(* Logix 5000 project; controller OT8 vendor 1 type 14 code 149 rev 32.11; software revision 32.04 *)

TASK MainTask (continuous, watchdog 500 ms) : MainProgram

MODULES
   Local : vendor 1 type 14 code 149 (Compact 0, rev 32.11)
      Discrete_IO : Embedded (Compact 1, rev 3.1, Output RPI 20 ms)
      VFD0602 : PowerFlex 525-EENET (Ethernet 100.100.100.11, rev 7.1, Output RPI 20 ms)
      VFD0543 : PowerFlex 525-EENET (Ethernet 100.100.100.10, rev 7.1, Output RPI 20 ms)
      VFD0643 : PowerFlex 525-EENET (Ethernet 100.100.100.12, rev 7.1, Output RPI 20 ms)
END_MODULES

TYPE VFD_CONTROL :
STRUCT
   START_CONDITION : BOOL;   // START CONDITIONS TRUE
   AUTO_RUN_VFD : BOOL;   // RUN VFD IN AUTO MODE
   VFD_RUNNING : BOOL;
   ALARM : BOOL;   // VFD ALARM WENT ACTIVE
   VFD_RUN_REFERENCE : REAL;   // VFD SPEED REFERENCE TO RUN
   SELECTION_SPEEDS_STORAGE : REAL[17];   // VFD STORED SPEED
   START_TIMER : TIMER;   // VFD START DELAY TIMER READY TO START
   VFD_FP : VFD_FACEPLATE_DATA;
   ALARM_LATCH : BOOL;   // LOCAL ROUTINE ALARM LATCH
END_STRUCT
END_TYPE

TYPE VFD_FACEPLATE_DATA :
STRUCT
   _0 : BOOL;   // HMI FACEPLATE SPEED CHANGE
   _1 : BOOL;   // HMI FACEPLATE DISCONNECT ON
   _2 : BOOL;   // HMI FACEPLATE DISCONNECT FAULTED
   _3 : BOOL;   // HMI FACEPLATE MCP FAULTED
   _4 : BOOL;   // HMI FACEPLATE VFD READY
   _5 : BOOL;   // HMI FACEPLATE VFD FAULTED
   _6 : BOOL;   // HMI FACEPLATE ACTIVE
   _7 : BOOL;   // HMI FACEPLATE VFD COMMS OK
   _8 : BOOL;   // HMI FACEPLATE JOG PB
   _9 : BOOL;   // HMI FACEPLATE JOGGING INDICATOR
   _10 : BOOL;   // HMI FACEPLATE SPARE At Reference Reached (latching)
   _11 : BOOL;   // HMI FACEPLATE AUTO ACTIVE
   _12 : BOOL;   // HMI FACEPLATE MANUAL RUN MODE ACTIVE
   SPARE1 : BOOL;
   SPARE2 : BOOL;
   SPARE3 : BOOL;
   HMI_SPEED_REF : REAL;   // VFD SPEED REFERENCE FROM HMI
   HMI_OUT_FREQ : REAL;   // VFD OUTPUT FREQUENCY TO HMI
   HMI_OUT_CUR : REAL;   // VFD OUTPUT CURRENT TO HMI
   SPEED_REF : REAL;   // VFD SELECTED SPEED REFERENCE
   COMMS_FAULT_CODE : DINT;   // .2 AND .9 HIGH = COMMS GOOD
END_STRUCT
END_TYPE

VAR_GLOBAL   (* controller tags *)
   ALARM_ACTIVE : BOOL;   // LINE 41 PLC ALARM BIT IS SET
   ALARMS : DINT[3];
        [0]   // VFD ALARMS
        [0].0   // VFD0543 NOT READY ALARM
        [0].1   // VFD0602 NOT READY ALARM
        [0].10   // VFD1043 NOT READY ALARM
        [0].11   // VFD1102 NOT READY ALARM
        [0].12   // VFD1143 NOT READY ALARM
        [0].13   // VFD1202 NOT READY ALARM
        [0].14   // VFD1243 NOT READY ALARM
        [0].2   // VFD0643 NOT READY ALARM
        [0].3   // VFD0702 NOT READY ALARM
        [0].4   // VFD0743 NOT READY ALARM
        [0].5   // VFD0802 NOT READY ALARM
        [0].6   // VFD0843 NOT READY ALARM
        [0].7   // VFD0902 NOT READY ALARM
        [0].8   // VFD0943 NOT READY ALARM
        [0].9   // VFD1002 NOT READY ALARM
        [1]   // DISC ALARMS
        [1].0   // DS0543 AUX CONTACT ALARM
        [1].1   // DS0602 AUX CONTACT ALARM
        [1].10   // DS1043 AUX CONTACT ALARM
        [1].11   // DS1102 AUX CONTACT ALARM
        [1].12   // DS1143 AUX CONTACT ALARM
        [1].13   // DS1202 AUX CONTACT ALARM
        [1].14   // DS1243 AUX CONTACT ALARM
        [1].2   // DS0643 AUX CONTACT ALARM
        [1].3   // DS0702 AUX CONTACT ALARM
        [1].4   // DS0743 AUX CONTACT ALARM
        [1].5   // DS0802 AUX CONTACT ALARM
        [1].6   // DS0808 AUX CONTACT ALARM
        [1].7   // DS0814 AUX CONTACT ALARM
        [1].8   // DS0943 AUX CONTACT ALARM
        [1].9   // DS1002 AUX CONTACT ALARM
        [2]   // E-STOP ALARMS
        [2].0   // E-STOP MAIN ENCLOSURE PBLT1402 ALARM
        [2].1   // E-STOP REMOTE #1 PBLT1404 ALARM
        [2].2   // E-STOP REMOTE #2 PBLT1406 ALARM
        [2].3   // E-STOP REMOTE #3 PBLT1408 ALARM
        [2].4   // E-STOP REMOTE #4 PBLT1410 ALARM
        [2].5   // E-STOP REMOTE #5PBLT1412 ALARM
        [2].6   // E-STOP REMOTE #6 PBLT1414 ALARM
   DS0543 : ALIAS FOR Local:1:I.Data.8;   // DS0543 AUX CONTACT
   DS0602 : ALIAS FOR Local:1:I.Data.9;   // DS0602 AUX CONTACT
   DS0643 : ALIAS FOR Local:1:I.Data.10;   // DS0643 AUX CONTACT
   LINE_100_RESET : ALIAS FOR Local:1:I.Data.6;   // LINE 100 RESET ALARMS
   LINE_100_RUN_MODE_ACTIVE : BOOL := 1;   // LINE 100 RUN MODE ACTIVE
   LINE_100_RUN_MODE_READY : BOOL := 1;   // LINE 100 IS READY TO START
   LINE_100_STARTUP_ANNUNCIATION_DELAY : TIMER := (PRE := 3000);   // LINE 100 STARTUP DELAY
   LINE_100_VFD_READY : BOOL := 1;   // LINE 100 VFDS READY
   LINE_200_RUN_MODE_ACTIVE : BOOL := 1;   // LINE 200 RUN MODE ACTIVE
   LINE_200_RUN_MODE_READY : BOOL := 1;   // LINE 200 IS READY TO START
   LINE_200_START_FLASH_BIT : BOOL;   // BIT TO FLASH LINE 200 START PB PILOT LIGHT DURING STARTUP
   LINE_200_STARTUP_ANNUNCIATION_DELAY : TIMER := (PRE := 3000);   // LINE 200 STARTUP DELAY
   LINE_200_VFD_READY : BOOL := 1;   // LINE 200 VFD READY
   LINE_200_VFDS_READY : BOOL;   // LINE 200 VFDS READY
   PB1831 : ALIAS FOR Local:1:I.Data.2;   // LINE 100 STOP PB
   PB1832 : ALIAS FOR Local:1:I.Data.3;   // LINE 100 START PB
   PB1833 : ALIAS FOR Local:1:I.Data.4;   // LINE 200 STOP PB
   PB1834 : ALIAS FOR Local:1:I.Data.5;   // LINE 200 START PB
   PBLT1832 : ALIAS FOR Local:1:O.Data.0;   // LINE 100 START PB PILOT LIGHT
   PBLT1834 : ALIAS FOR Local:1:O.Data.1;   // LINE 200 START PB PILOT LIGHT
   SAFETY_RELAY_RESET_ONS : BOOL;
   SR1426 : ALIAS FOR Local:1:I.Data.0;   // LINE 200 SAFETY RELAY
   SR1526 : ALIAS FOR Local:1:I.Data.1;   // LINE 100 SAFETY RELAY
   STARTUP_ANNUNCIATION_DELAY : TIMER;   // STARTUP ANNUCIATION TIMER
   SYSTEM_AUTO_RUN_MODE_ACTIVE : BOOL;   // RUN MODE ACTIVE
   SYSTEM_AUTO_RUN_MODE_READY : BOOL;   // SYSTEM READY TO ENTER AUTO RUN MODE
   SYSTEM_FLASH_BIT : BOOL := 1;   // FLASH BIT
   SYSTEM_FLASHER_OFF_TIME : TIMER := (PRE := 500, ACC := 500);   // SYSTEM FLASHER OFF TIME
   SYSTEM_FLASHER_ON_TIME : TIMER := (PRE := 500, ACC := 19, EN := 1, TT := 1);   // SYSTEM FLASHER ON TIME
   VFD0543 : VFD_CONTROL := (START_CONDITION := 1, START_TIMER.PRE := 500, START_TIMER.ACC := 500, START_TIMER.EN := 1, START_TIMER.DN := 1);
   VFD0602 : VFD_CONTROL := (START_CONDITION := 1, START_TIMER.PRE := 500, START_TIMER.ACC := 500, START_TIMER.EN := 1, START_TIMER.DN := 1);
   VFD0643 : VFD_CONTROL := (START_CONDITION := 1, START_TIMER.EN := 1, START_TIMER.DN := 1);
END_VAR

PROGRAM MainProgram   (* main routine MainRoutine *)
VAR
   AFI : DINT;
   PBLT1437 : ALIAS FOR Local:1:I.Data.6;   // RESET PUSHBUTTON LINE 200
   PBLT1537 : ALIAS FOR Local:1:I.Data.7;   // RESET PUSHBUTTON LINE 100
END_VAR

ROUTINE ALARMS   (* ladder *)
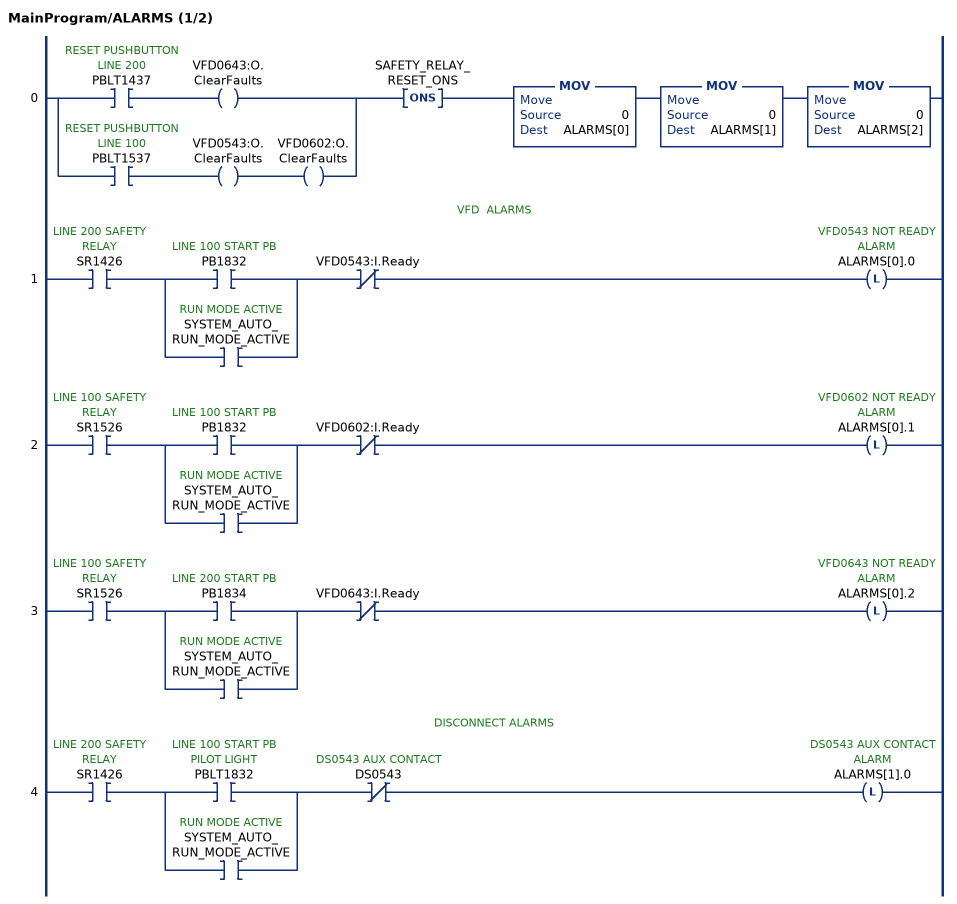
   0: [XIC(PBLT1437) OTE(VFD0643:O.ClearFaults) ,XIC(PBLT1537) OTE(VFD0543:O.ClearFaults) OTE(VFD0602:O.ClearFaults) ]ONS(SAFETY_RELAY_RESET_ONS)MOV(0,ALARMS[0])MOV(0,ALARMS[1])MOV(0,ALARMS[2]);
   // VFD  ALARMS
   1: XIC(SR1426)[XIC(PB1832) ,XIC(SYSTEM_AUTO_RUN_MODE_ACTIVE) ]XIO(VFD0543:I.Ready)OTL(ALARMS[0].0);
   2: XIC(SR1526)[XIC(PB1832) ,XIC(SYSTEM_AUTO_RUN_MODE_ACTIVE) ]XIO(VFD0602:I.Ready)OTL(ALARMS[0].1);
   3: XIC(SR1526)[XIC(PB1834) ,XIC(SYSTEM_AUTO_RUN_MODE_ACTIVE) ]XIO(VFD0643:I.Ready)OTL(ALARMS[0].2);
   // DISCONNECT ALARMS
   4: XIC(SR1426)[XIC(PBLT1832) ,XIC(SYSTEM_AUTO_RUN_MODE_ACTIVE) ]XIO(DS0543)OTL(ALARMS[1].0);
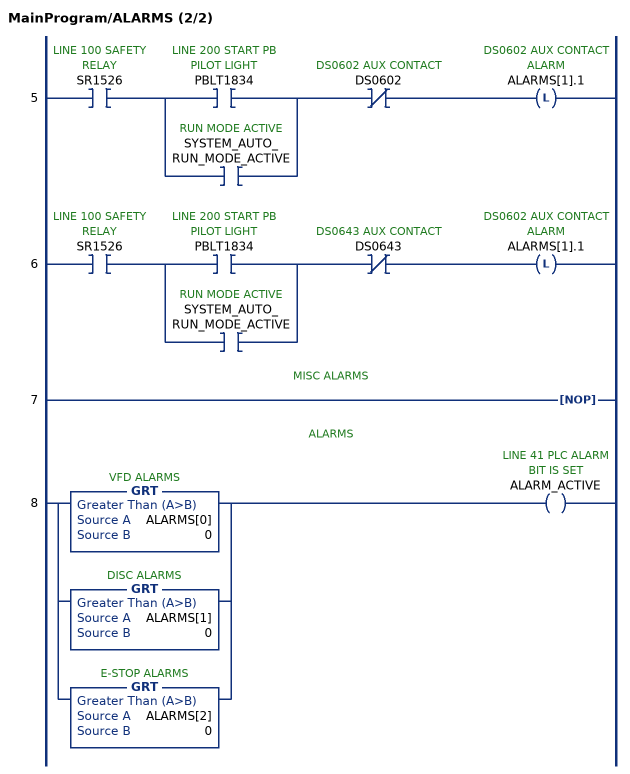
   5: XIC(SR1526)[XIC(PBLT1834) ,XIC(SYSTEM_AUTO_RUN_MODE_ACTIVE) ]XIO(DS0602)OTL(ALARMS[1].1);
   6: XIC(SR1526)[XIC(PBLT1834) ,XIC(SYSTEM_AUTO_RUN_MODE_ACTIVE) ]XIO(DS0643)OTL(ALARMS[1].1);
   // MISC ALARMS
   7: NOP();
   // ALARMS
   8: [GRT(ALARMS[0],0) ,GRT(ALARMS[1],0) ,GRT(ALARMS[2],0) ]OTE(ALARM_ACTIVE);
END_ROUTINE

ROUTINE MainRoutine   (* ladder *)
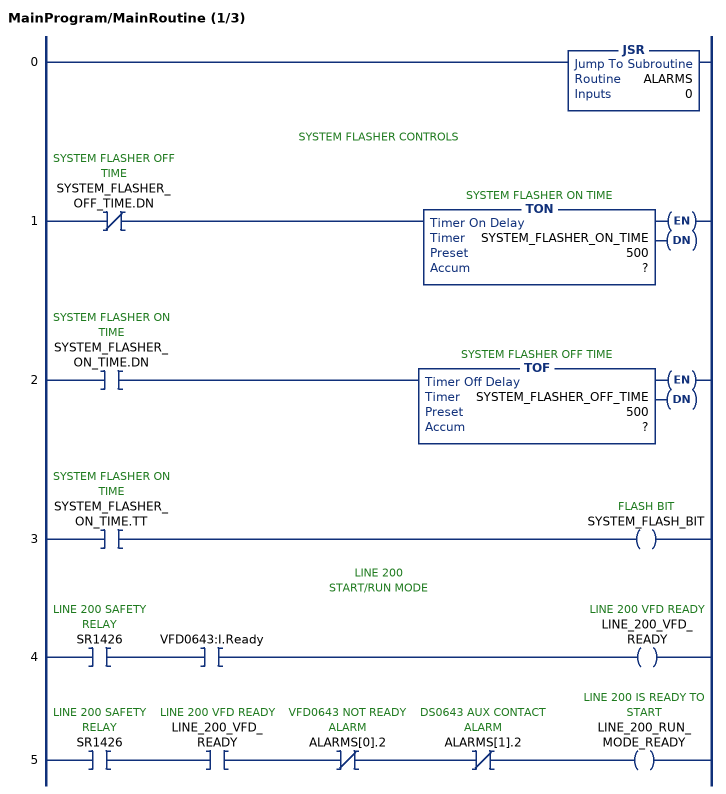
   0: JSR(ALARMS,0);
   // SYSTEM FLASHER CONTROLS
   1: XIO(SYSTEM_FLASHER_OFF_TIME.DN)TON(SYSTEM_FLASHER_ON_TIME,?,?);
   2: XIC(SYSTEM_FLASHER_ON_TIME.DN)TOF(SYSTEM_FLASHER_OFF_TIME,?,?);
   3: XIC(SYSTEM_FLASHER_ON_TIME.TT)OTE(SYSTEM_FLASH_BIT);
   // LINE 200
   // START/RUN MODE
   4: XIC(SR1426)XIC(VFD0643:I.Ready)OTE(LINE_200_VFD_READY);
   5: XIC(SR1426)XIC(LINE_200_VFD_READY)XIO(ALARMS[0].2)XIO(ALARMS[1].2)OTE(LINE_200_RUN_MODE_READY);
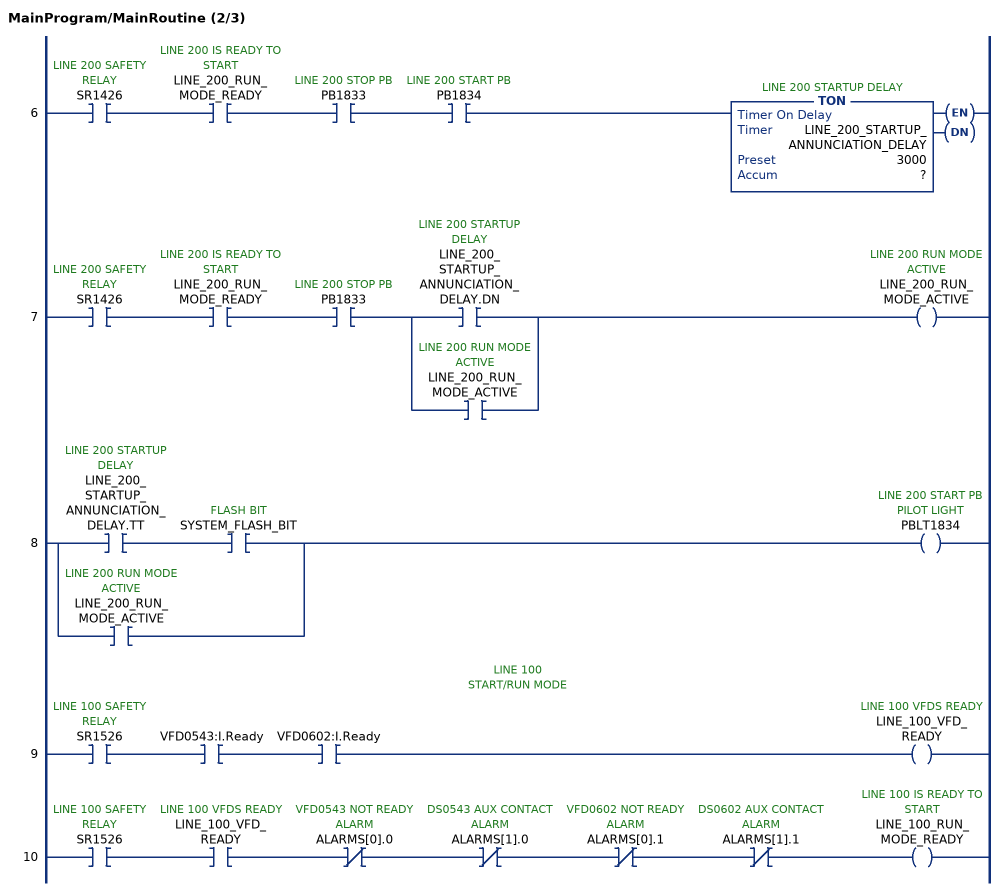
   6: XIC(SR1426)XIC(LINE_200_RUN_MODE_READY)XIC(PB1833)XIC(PB1834)TON(LINE_200_STARTUP_ANNUNCIATION_DELAY,?,?);
   7: XIC(SR1426)XIC(LINE_200_RUN_MODE_READY)XIC(PB1833)[XIC(LINE_200_STARTUP_ANNUNCIATION_DELAY.DN) ,XIC(LINE_200_RUN_MODE_ACTIVE) ]OTE(LINE_200_RUN_MODE_ACTIVE);
   8: [XIC(LINE_200_STARTUP_ANNUNCIATION_DELAY.TT) XIC(SYSTEM_FLASH_BIT) ,XIC(LINE_200_RUN_MODE_ACTIVE) ]OTE(PBLT1834);
   // LINE 100
   // START/RUN MODE
   9: XIC(SR1526)XIC(VFD0543:I.Ready)XIC(VFD0602:I.Ready)OTE(LINE_100_VFD_READY);
   10: XIC(SR1526)XIC(LINE_100_VFD_READY)XIO(ALARMS[0].0)XIO(ALARMS[1].0)XIO(ALARMS[0].1)XIO(ALARMS[1].1)OTE(LINE_100_RUN_MODE_READY);
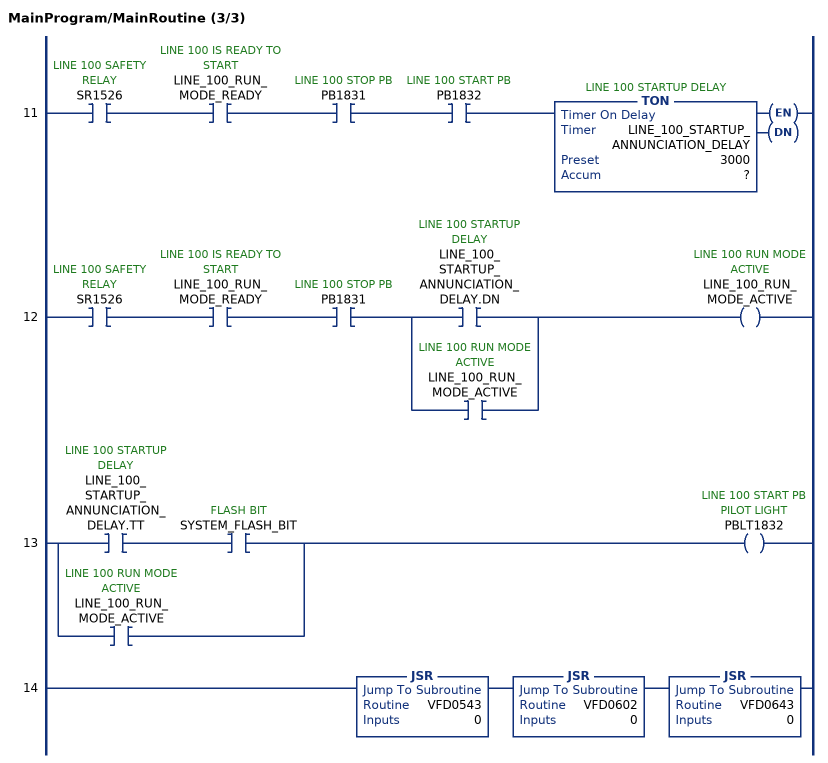
   11: XIC(SR1526)XIC(LINE_100_RUN_MODE_READY)XIC(PB1831)XIC(PB1832)TON(LINE_100_STARTUP_ANNUNCIATION_DELAY,?,?);
   12: XIC(SR1526)XIC(LINE_100_RUN_MODE_READY)XIC(PB1831)[XIC(LINE_100_STARTUP_ANNUNCIATION_DELAY.DN) ,XIC(LINE_100_RUN_MODE_ACTIVE) ]OTE(LINE_100_RUN_MODE_ACTIVE);
   13: [XIC(LINE_100_STARTUP_ANNUNCIATION_DELAY.TT) XIC(SYSTEM_FLASH_BIT) ,XIC(LINE_100_RUN_MODE_ACTIVE) ]OTE(PBLT1832);
   14: JSR(VFD0543,0)JSR(VFD0602,0)JSR(VFD0643,0);
END_ROUTINE

ROUTINE VFD0543   (* ladder *)
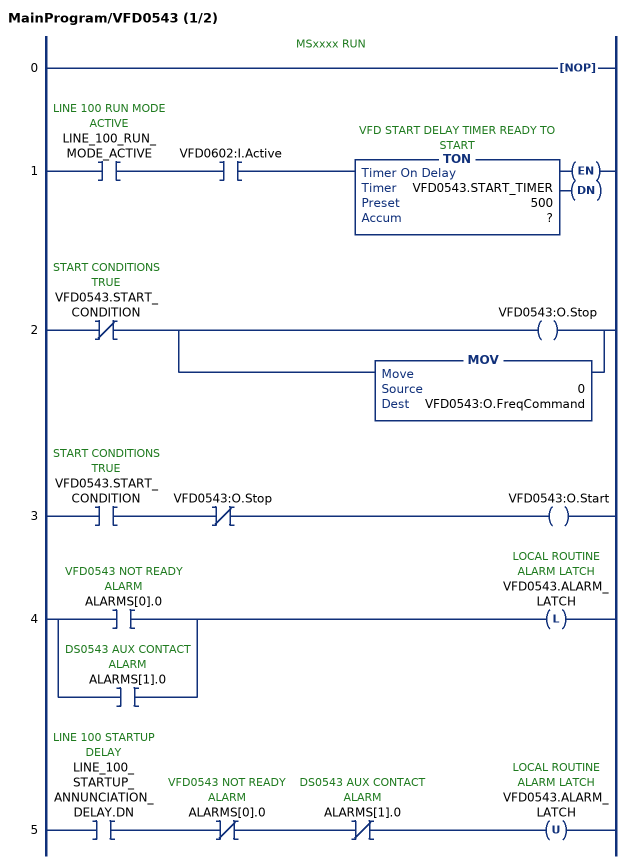
   // MSxxxx RUN
   0: NOP();
   1: XIC(LINE_100_RUN_MODE_ACTIVE)XIC(VFD0602:I.Active)TON(VFD0543.START_TIMER,?,?);
   2: XIO(VFD0543.START_CONDITION)[OTE(VFD0543:O.Stop) ,MOV(0,VFD0543:O.FreqCommand) ];
   3: XIC(VFD0543.START_CONDITION)XIO(VFD0543:O.Stop)OTE(VFD0543:O.Start);
   4: [XIC(ALARMS[0].0) ,XIC(ALARMS[1].0) ]OTL(VFD0543.ALARM_LATCH);
   5: XIC(LINE_100_STARTUP_ANNUNCIATION_DELAY.DN)XIO(ALARMS[0].0)XIO(ALARMS[1].0)OTU(VFD0543.ALARM_LATCH);
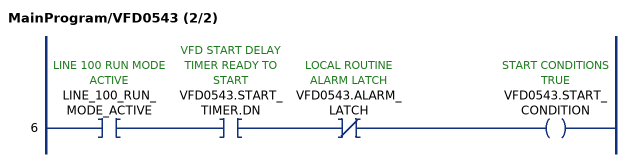
   6: XIC(LINE_100_RUN_MODE_ACTIVE)XIC(VFD0543.START_TIMER.DN)XIO(VFD0543.ALARM_LATCH)OTE(VFD0543.START_CONDITION);
END_ROUTINE

ROUTINE VFD0602   (* ladder *)
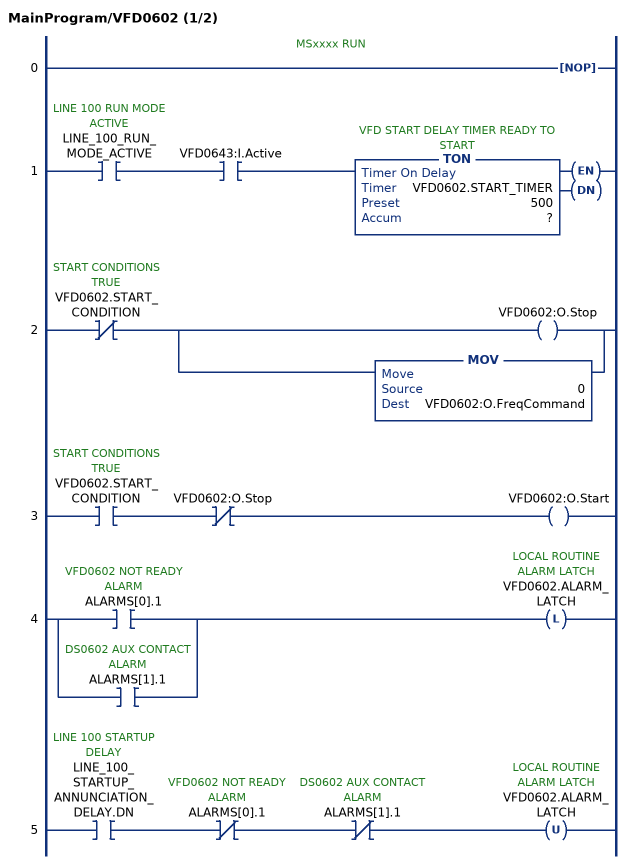
   // MSxxxx RUN
   0: NOP();
   1: XIC(LINE_100_RUN_MODE_ACTIVE)XIC(VFD0643:I.Active)TON(VFD0602.START_TIMER,?,?);
   2: XIO(VFD0602.START_CONDITION)[OTE(VFD0602:O.Stop) ,MOV(0,VFD0602:O.FreqCommand) ];
   3: XIC(VFD0602.START_CONDITION)XIO(VFD0602:O.Stop)OTE(VFD0602:O.Start);
   4: [XIC(ALARMS[0].1) ,XIC(ALARMS[1].1) ]OTL(VFD0602.ALARM_LATCH);
   5: XIC(LINE_100_STARTUP_ANNUNCIATION_DELAY.DN)XIO(ALARMS[0].1)XIO(ALARMS[1].1)OTU(VFD0602.ALARM_LATCH);
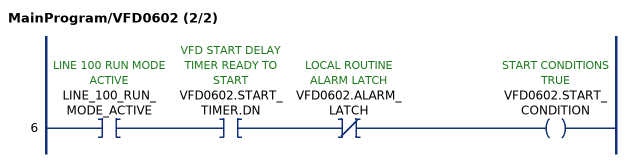
   6: XIC(LINE_100_RUN_MODE_ACTIVE)XIC(VFD0602.START_TIMER.DN)XIO(VFD0602.ALARM_LATCH)OTE(VFD0602.START_CONDITION);
END_ROUTINE

ROUTINE VFD0643   (* ladder *)
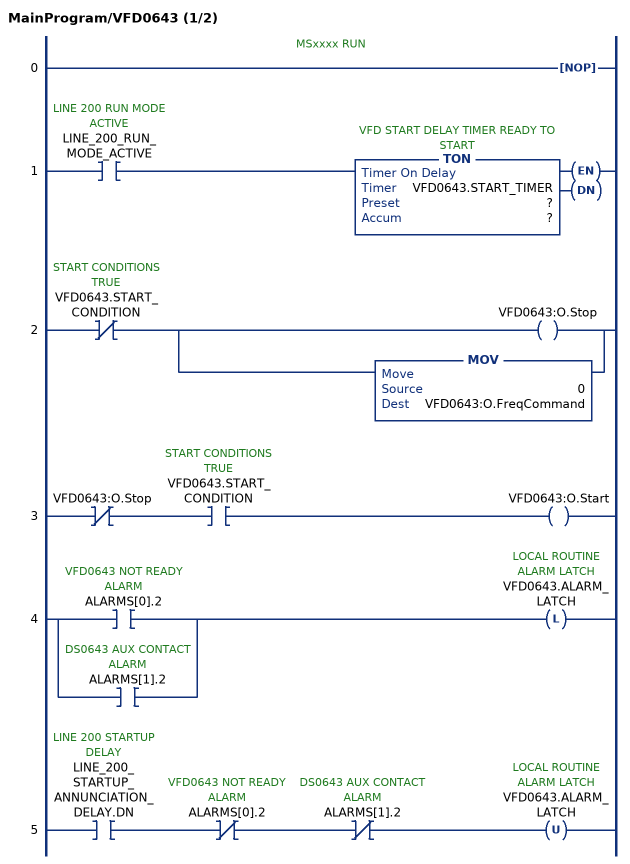
   // MSxxxx RUN
   0: NOP();
   1: XIC(LINE_200_RUN_MODE_ACTIVE)TON(VFD0643.START_TIMER,?,?);
   2: XIO(VFD0643.START_CONDITION)[OTE(VFD0643:O.Stop) ,MOV(0,VFD0643:O.FreqCommand) ];
   3: XIO(VFD0643:O.Stop)XIC(VFD0643.START_CONDITION)OTE(VFD0643:O.Start);
   4: [XIC(ALARMS[0].2) ,XIC(ALARMS[1].2) ]OTL(VFD0643.ALARM_LATCH);
   5: XIC(LINE_200_STARTUP_ANNUNCIATION_DELAY.DN)XIO(ALARMS[0].2)XIO(ALARMS[1].2)OTU(VFD0643.ALARM_LATCH);
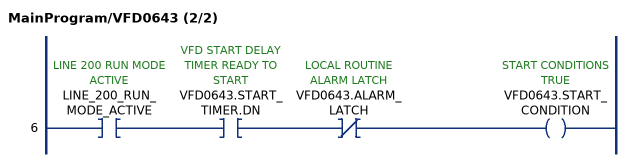
   6: XIC(LINE_200_RUN_MODE_ACTIVE)XIC(VFD0643.START_TIMER.DN)XIO(VFD0643.ALARM_LATCH)OTE(VFD0643.START_CONDITION);
END_ROUTINE
END_PROGRAM
